FUNCTION_BLOCK FB_Camera
(*
********************************************************************************
* Name: FB_Camera
*
* Author:  AutomanH
* Version: 1.0.0
*
* Description:
*	Camera trigger and camera lights control
*
* Remarks:
*
*
* Revisions:
*   V1.0.0 -Automanh 2022.06.08
*		V2.0.0-Automanh 2022.07.15 add Timeout Error and xQDone Single
*********************************************************************************)
VAR_INPUT
	xlInit	:BOOL;(*初始化*)
	xlTrigger:BOOL;(*相机触发*)
	xlTriggerHmi:BOOL;(*触摸屏相机触发*)
	xlLight  :BOOL;(*是否存在光源*)
	xlReady	 :BOOL;(*相机准备就绪信号*)
	xlAutoMode:BOOL;(*自动模式*)
	xlManualMode:BOOL;(*手动模式*)
	xITryRun:BOOL;(*空跑*)
	tlDelay: TIME;  (*打开光源与拍照间隔的时间*)
	xIDeviceRunning :BOOL;(*单循环运行*)
	
END_VAR
VAR_OUTPUT
	xQStart	:BOOL;			//开始拍照
	xQLight: BOOL := FALSE;//打开光源
	xQCompleted:BOOL;		//拍照完成
	xQAlarm	: BOOL := FALSE;// 报警输出
	xQBusy	 	:BOOL;
	xQHmiAlarm	:STRING;//报警输出
	xQDone	  :BOOL;
END_VAR
VAR_IN_OUT
	ilCompleted :INT;(*拍照完成*)
END_VAR
VAR
	bStep:BYTE;
	{attribute 'hide'}
	tonDelay: TON;//计时器
	{attribute 'hide'}
	tonAlarmTime :Ton;//报警计时器
	{attribute 'hide'}
	tTimeout:TON;
END_VAR

ACT_Init();
ACT_Trigger();
ACT_Alarm();

ACTION ACT_Alarm:
IF NOT xlReady THEN
	xQHmiAlarm:='Not Ready';
ELSIF xlReady AND NOT xQBusy THEN
 	xQHmiAlarm:='Ready';
ELSIF xQAlarm THEN
	xQHmiAlarm:='Time out';
END_IF
END_ACTION

ACTION ACT_Init:
IF  xlInit THEN
	xlTrigger:=FALSE;	
	xlTriggerHmi:=FALSE;
	xlLight :=FALSE;
	ilCompleted:=0;
	xQStart:=FALSE;
	xQLight:=FALSE;
	xQCompleted:=FALSE;
	xQAlarm	  :=FALSE;
	xQBusy    :=FALSE;
	xQDone		:=FALSE;
	xlInit	  :=FALSE;
END_IF
END_ACTION

ACTION ACT_Trigger:

CASE bStep OF
	0://等待触发
		tonDelay(IN:=FALSE);
		tonAlarmTime(IN:=FALSE);
		ilCompleted:=0;
		IF (( (xlAutomode OR xIDeviceRunning) AND xlTrigger) OR
				(xlManualmode AND xlTriggerHmi)) AND (xlReady OR xITryRun) THEN
			xlTrigger:=xlTriggerHmi:=FALSE;
			xQCompleted:=FALSE;
			xQBusy:=TRUE;
			xQDone:=FALSE;
			bStep:=bStep +1;
		END_IF
	
	1://打开光源信号
		 IF  NOT xITryRun THEN
			 IF xlLight THEN
				 xQLight:=TRUE;
			 END_IF
		 END_IF
			 bStep:=bStep+1;		
	2://开始拍照
		IF  NOT   xITryRun THEN
			 tonDelay(IN:=TRUE,PT:=tlDelay,	Q=>,ET=>);
			 IF  tonDelay.Q  THEN
				 xQStart:=TRUE;
				 xQHmiAlarm:='Started';
				 tonDelay(IN:=FALSE);
				 bStep:=bStep+1;		
			 END_IF
		ELSE
				bStep:=bStep+1;		
		END_IF
 3://拍照结束
	 		IF  ilCompleted = 1 OR xITryRun THEN 
			 	ilCompleted:=0;
			 	xQStart:=FALSE;
				xQLight:=FALSE;
				bStep:=bStep+1;	
				xQCompleted:=TRUE;	
			ELSE
				tonAlarmTime(IN:=TRUE,PT:=T#3S,	Q=>,ET=>);
				IF    tonAlarmTime.Q THEN
				 	xQStart:=FALSE;
					xQLight:=FALSE;
					xQAlarm:=TRUE;
					tonAlarmTime(IN:=FALSE);
					bStep:=0;	
				END_IF
			END_IF
	4://关闭光源
			xQCompleted:=TRUE;
			xQLight:=FALSE;
			bStep:=bStep+1;	
	5://流程结束
			xQHmiAlarm:='Completed';
			xQBusy:=FALSE;
			xQDone:=TRUE;
			bStep:=0;	
END_CASE
END_ACTION

END_FUNCTION_BLOCK

(* stored: Version 1.1.0.1, ProductVersion 3.1.4024.9
   POU FB_Camera: Id {d6929595-da25-4baa-b108-0d912ac90d24}, SpecialFunc None
   Action ACT_Alarm: Id {42165045-1927-44c9-8eee-258a82b0f70d}
   Action ACT_Init: Id {4b8c9287-3be3-4a47-a770-80413c4d9c30}
   Action ACT_Trigger: Id {9183c163-8be5-4fbe-86c9-2c27dadf0cba} *)
